// TIA Portal V17 export
// export: Created 2025-03-05T08:00:54.6070687Z, ExportSetting WithDefaults, DisplayName Totally Integrated Automation Portal, DisplayVersion V17 Update 8, DisplayName TIA Portal Openness, DisplayVersion V17 Update 8, DisplayName TIA Portal Version Control Interface, DisplayVersion V17, DisplayName SINAMICS Startdrive Advanced, DisplayVersion V17 SP2, DisplayName SINAMICS Startdrive G110M, G120, G120C, G120D, G120P, G115D, DisplayVersion V17 SP2, DisplayName SINAMICS Startdrive G130, G150, S120, S150, SINAMICS MV, S210, DisplayVersion V17 SP2, DisplayName STEP 7 Professional, DisplayVersion V17 Update 8, DisplayName SINUMERIK ONE STEP 7 Toolbox, DisplayVersion V17 Update 12, DisplayName SINUMERIK 840D sl STEP 7 Toolbox, DisplayVersion V17 Update 12, DisplayName STEP 7 Safety, DisplayVersion V17 Update 6, DisplayName WinCC Advanced, DisplayVersion V17 Update 8
DATA_BLOCK "DB1472_UNIT_02_LASER_COOLING_ALARMS"   // DB1472
{ DB_Accessible_From_OPC_UA := 'FALSE' }
AUTHOR : ETXETAR
VERSION : 1.0
// stored: AutoNumber false, DBAccessibleFromOPCUA false, DBAccessibleFromWebserver true, InstanceOfName FB1453_LASER_COOLING_ALARMS, InstanceOfType FB
"FB1453_LASER_COOLING_ALARMS"
   // VAR_INPUT
   //    OPTIONS_0 : Byte;
   //    OPTIONS_1 : Byte;
   //    LASER_OUTPUT_FLOW_LOW_VALUE_ALM_BIT : Bool;
   //    NOZZLE_FLOW_LOW_VALUE_ALM_BIT : Bool;
   //    HEAD_FLOW_LOW_VALUE_ALM_BIT : Bool;
   //    LASER_OUTPUT_OVERTEMPERATURE_ALM_BIT : Bool;
   //    NOZZLE_OVERTEMPERATURE_ALM_BIT : Bool;
   //    HEAD_OVERTEMPERATURE_ALM_BIT : Bool;
   //    LASER_OUTPUT_FLOW_RAW_INPUT : DInt;
   //    LASER_OUTPUT_TEMP_RAW_INPUT : DInt;
   //    NOZZLE_COOLING_FLOW_RAW_INPUT : Word;
   //    NOZZLE_COOLING_TEMP_RAW_INPUT : Word;
   //    HEAD_COOLING_FLOW_RAW_INPUT : DInt;
   //    HEAD_COOLING_TEMP_RAW_INPUT : DInt;
   //    LASER_READY : Bool;
   //    UNIT_ALARM : UInt;
   // END_VAR
   // VAR_OUTPUT
   //    OUTPUT_LOW_FLOW_ALARM : Bool;
   //    OUTPUT_HIGH_FLOW_ALARM : Bool;
   //    OUTPUT_FLOW_SETPOINT_ALARM : Bool;
   //    OUTPUT_LOW_TEMP_ALARM : Bool;
   //    OUTPUT_HIGH_TEMP_ALARM : Bool;
   //    OUTPUT_TEMP_SETPOINT_ALARM : Bool;
   //    NOZZLE_LOW_FLOW_ALARM : Bool;
   //    NOZZLE_HIGH_FLOW_ALARM : Bool;
   //    NOZZLE_FLOW_SETPOINT_ALARM : Bool;
   //    NOZZLE_LOW_TEMP_ALARM : Bool;
   //    NOZZLE_HIGH_TEMP_ALARM : Bool;
   //    NOZZLE_TEMP_SETPOINT_ALARM : Bool;
   //    HEAD_LOW_FLOW_ALARM : Bool;
   //    HEAD_HIGH_FLOW_ALARM : Bool;
   //    HEAD_FLOW_SETPOINT_ALARM : Bool;
   //    HEAD_LOW_TEMP_ALARM : Bool;
   //    HEAD_HIGH_TEMP_ALARM : Bool;
   //    HEAD_TEMP_SETPOINT_ALARM : Bool;
   //    OUTPUT_LOW_FLOW_WARNING : Bool;
   //    OUTPUT_HIGH_FLOW_WARNING : Bool;
   //    OUTPUT_LOW_TEMP_WARNING : Bool;
   //    OUTPUT_HIGH_TEMP_WARNING : Bool;
   //    NOZZLE_LOW_FLOW_WARNING : Bool;
   //    NOZZLE_HIGH_FLOW_WARNING : Bool;
   //    NOZZLE_LOW_TEMP_WARNING : Bool;
   //    NOZZLE_HIGH_TEMP_WARNING : Bool;
   //    HEAD_LOW_FLOW_WARNING : Bool;
   //    HEAD_HIGH_FLOW_WARNING : Bool;
   //    HEAD_LOW_TEMP_WARNING : Bool;
   //    HEAD_HIGH_TEMP_WARNING : Bool;
   // END_VAR
   // VAR RETAIN
   //    ANY_ACTIVE_ALARM : Bool;
   //    RHP_SEOC_ALARMS : Bool;
   //    IS_SEOC_ALARMS : Bool;
   //    WARNINGS : Bool;
   //    WARNINGS_GONE : Bool;
   //    COOLING_ALARMS_ENABLED : Bool;
   //    LASER_OUTPUT_SENSOR_VALUES { ExternalAccessible := 'False'; ExternalVisible := 'False'; ExternalWritable := 'False'} : "COOLING_SENSOR";
   //    NOZZLE_SENSOR_VALUES { ExternalAccessible := 'False'; ExternalVisible := 'False'; ExternalWritable := 'False'} : "COOLING_SENSOR";
   //    LASER_HEAD_SENSOR_VALUES { ExternalAccessible := 'False'; ExternalVisible := 'False'; ExternalWritable := 'False'} : "COOLING_SENSOR";
   // END_VAR
BEGIN
END_DATA_BLOCK
